ABB RobotStudio station: RWS_simple_RW6.16.rspag

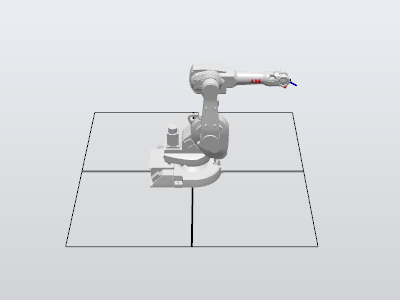
--- station ---
Station RWS_simple_RW6.16 (saved by RobotStudio 25.3.11371.0)
Controller IRB1600_6_120
  mechanical unit ROB_1: IRB1600_6_120__03, 6 joints, base frame (0, 0, 0) mm
Layout (positions relative to the parent item):
  - IRB1600_6_120__03 [mechanism, from %ABB.RobotStudio.Models.IRB1600%\IRB1600_6_120_G_03.rslib] at (0, 0, 0) mm; joint values [0, 0, 0, 0, 0.5236, 0] (rad or m)

--- Controller Data/IRB1600_6_120/RAPID/TASK1/PROGMOD/MainModule.mod ---
MODULE MainModule
    VAR num nCounter;

    PROC main()
        WaitTime 5;
    ENDPROC
ENDMODULE

--- Controller Data/IRB1600_6_120/SYSPAR/EIO.cfg ---
EIO:CFG_1.0:6:1::
#
INDUSTRIAL_NETWORK:

      -Name "DeviceNet" -Label "DeviceNet Master/Slave Network" -Address "2"
#
DEVICENET_INTERNAL_DEVICE:

      -Name "DN_Internal_Device" -VendorName "ABB Robotics"\
      -ProductName "DeviceNet Internal Slave Device"
#
EIO_SIGNAL:

      -Name "DI1" -SignalType "DI" -Device "DN_Internal_Device" -DeviceMap "1"

      -Name "DO1" -SignalType "DO" -Device "DN_Internal_Device" -DeviceMap "1"\
      -Access "All"
